PROGRAM MAIN
VAR
a : INT;
b : INT;
c : INT;

END_VAR

c := a+b;

END_PROGRAM

(* stored: Version 1.1.0.1, ProductVersion 3.1.4024.4
   POU MAIN: Id {a9ed13f8-7010-4aa8-be47-ba11eca525c0}, SpecialFunc None *)
